(* CoDeSys 2.3.9.28 project: Codesys_Automacao.pro *)
(* Libraries: Standard.lib 27.1.09 11:27:38, Util.lib 27.1.09 11:27:38, IecSfc.lib 24.11.08 08:07:15, SysLibTime.lib 27.1.09 11:27:38, SysTaskInfo.lib 24.11.08 08:07:15, SYSLIBCALLBACK.LIB 27.1.09 11:27:38 *)

(* PLC configuration (modules and I/O channels)
Hexswitch AT %IB0 [HexSwitch] rotary switch 0 = STOP, 1-15 = RUN
IOModules [CPX_MASTER] node 0, in %IB4 out %QB0
  8DI/8DO [CPX-8DI_8DO_Multi_I_O_module_1] node 0, in %IB4 out %QB0 {StringParam = 4,8,1,8,1; ByteParam = 7; ByteParam = 81; ByteParam = 0; ByteParam = 0; ByteParam = 0; ByteParam = 0; ByteParam = 0; IdleStateParam = 0; IdleModeParam = 255; IdleStateParam = 0; IdleModeParam = 255; IdleStateParam = 0; IdleModeParam = 255; IdleStateParam = 0; IdleModeParam = 255}
    AT %IB4 [ByteInput] -
    AT %QB0 [ByteOutput] -
  8DI/8DO [CPX-8DI_8DO_Multi_I_O_module_1] node 1, in %IB8 out %QB4 {StringParam = 4,8,1,8,1; ByteParam = 7; ByteParam = 81; ByteParam = 0; ByteParam = 0; ByteParam = 0; ByteParam = 0; ByteParam = 0; IdleStateParam = 0; IdleModeParam = 255; IdleStateParam = 0; IdleModeParam = 255; IdleStateParam = 0; IdleModeParam = 255; IdleStateParam = 0; IdleModeParam = 255}
    AT %IB8 [ByteInput] -
    AT %QB4 [ByteOutput] -
*)

(* Global variable list: Global_Variables *)
VAR_GLOBAL

	START AT %IX2.0 : BOOL;
	STOP AT %IX2.1 : BOOL;
	B0 AT %IX2.2 : BOOL;

	S1 AT %IX4.4 : BOOL;
	S2 AT %IX4.5 : BOOL;

	S3 AT %IX2.4 : BOOL;
	S4 AT %IX2.5 : BOOL;
	S5 AT %IX2.3 : BOOL;
	S6 AT %IX2.6 : BOOL;
	S7 AT %IX2.7 : BOOL;

	P2_IDA AT %QX2.0 : BOOL;
	P2_VOLTA AT %QX2.1 : BOOL;
	P1 AT %QX2.2 : BOOL;
	P3 AT %QX2.3 : BOOL;



	M1 AT %QX0.0 : BOOL;
	M2 AT %QX0.1 : BOOL;

	LP_1 AT %QX0.2 : BOOL;
	LP_2 AT %QX0.3 : BOOL;
	LP_3 AT %QX0.4 : BOOL;
	AL AT %QX0.5 : BOOL;




	PV_CONT_ENT : INT :=1;
	PV_CONT_SAI : INT :=1;


	M_START : BOOL;
	M_CONT: BOOL;
	M_P1: BOOL;
	M_TEMPERA: BOOL;
	M_2_ENT : BOOL;
	M_2_SAI : BOOL;
	M_ALARME: BOOL;

	MT_1 : BOOL;
	MT_2 : BOOL;
	MT_3 : BOOL;
	MT_4 : BOOL;
	MT_5 : BOOL;

	T_TEMPERA : TON;
	T_ALARME : TON;

    CONT_2_ENT: CTU;
	CONT_2_SAI : CTU;

	BUZZER : APITA_BUZZER;



END_VAR

(* POU PLC_PRG, ST *)
PROGRAM PLC_PRG
VAR

END_VAR
T_TEMPERA(IN:=M_TEMPERA,PT:=T#3S);
T_ALARME(IN:=M_ALARME,PT:=T#5500MS);

CONT_2_ENT(CU:= M_CONT, RESET:= M_2_ENT OR STOP, PV:= PV_CONT_ENT);
CONT_2_SAI(CU:= S7 AND MT_5, RESET:= M_2_SAI OR STOP, PV:= PV_CONT_SAI);

BUZZER(LIGA := AL, DESLIGA := T_ALARME.Q OR START);


IF B0 AND NOT M_START THEN
	PV_CONT_ENT := 1;
	PV_CONT_SAI := 1;
	LP_3 := TRUE;
END_IF

IF NOT B0 AND NOT M_START THEN
	PV_CONT_ENT := 3;
	PV_CONT_SAI := 3;
	LP_3 := FALSE;
END_IF


IF START THEN
	M_START:=TRUE;
	P2_VOLTA:=TRUE;
	LP_1:=TRUE;
END_IF


IF M_START AND S1 THEN
	M1:=TRUE;
	MT_1:=TRUE;
END_IF


IF S2 AND MT_1 THEN
	M_CONT:=TRUE;
	M1:=FALSE;
	MT_1:=FALSE;
ELSE
	M_CONT:= FALSE;
END_IF


IF CONT_2_ENT.Q THEN
	M1:=FALSE;
	P1:=TRUE;
	MT_2:=TRUE;
END_IF


IF S3 AND MT_2 THEN
	P2_IDA:=TRUE;
	P2_VOLTA:=FALSE;
	M_2_ENT:=TRUE;
	MT_2:=FALSE;
	MT_3:=TRUE;
END_IF


IF S4 AND M_2_ENT AND MT_3 THEN
	P2_IDA:=FALSE;
	P2_VOLTA:=TRUE;
	P1:=FALSE;
	MT_3:=FALSE;
	MT_4:=TRUE;
END_IF


IF S5 AND S6 AND MT_4 THEN
	M2:=TRUE;
	M_TEMPERA:=TRUE;
	MT_4:=FALSE;
END_IF


IF T_TEMPERA.Q THEN
	M2:=FALSE;
	P3:=TRUE;
	MT_5:=TRUE;
	LP_2:=TRUE;
END_IF


IF AL THEN
	M_ALARME :=TRUE;
END_IF


IF T_ALARME.Q THEN
	M_ALARME :=FALSE;
END_IF


IF CONT_2_SAI.Q THEN
	AL:=TRUE;
	M_2_ENT:=FALSE;
	M_2_SAI:=TRUE;
	M1:=FALSE;
	M2:=FALSE;

	P1:=FALSE;
	P2_IDA:=FALSE;
	P2_VOLTA:=FALSE;
	P3:=FALSE;

	M_TEMPERA:=FALSE;
	M_START:=FALSE;
	M_CONT:=FALSE;

	MT_1:=FALSE;
	MT_2:=FALSE;
	MT_3:=FALSE;
	MT_4:=FALSE;
	MT_5:=FALSE;

	LP_2:=FALSE;
	LP_1:=FALSE;
ELSE
	M_2_SAI:=FALSE;
END_IF


IF STOP THEN
	M_2_ENT:=FALSE;
	M_2_SAI:=FALSE;
	M_START:=FALSE;
	M1:=FALSE;
	M2:=FALSE;

	P1:=FALSE;
	P2_IDA:=FALSE;
	P2_VOLTA:=TRUE;
	P3:=FALSE;

	M_TEMPERA:=FALSE;
	M_START:=FALSE;
	M_CONT:=FALSE;

	MT_1:=FALSE;
	MT_2:=FALSE;
	MT_3:=FALSE;
	MT_4:=FALSE;
	MT_5:=FALSE;

	LP_2:=FALSE;
	LP_1:=FALSE;
	AL:=FALSE;
END_IF
END_PROGRAM

(* POU APITA_BUZZER, ST *)
FUNCTION_BLOCK APITA_BUZZER
VAR_INPUT
	LIGA : BOOL;
	DESLIGA : BOOL;
END_VAR
VAR_OUTPUT
	SAIDA : BOOL;
END_VAR
VAR
	T1 : TON;
	T2 : TON;
	MEM : BOOL;
END_VAR
T1(IN:=AL, PT:=T#500MS);
T2(IN:= NOT AL, PT:=T#500MS);

IF LIGA AND T1.Q AND MEM THEN
	AL := FALSE;
END_IF


IF NOT LIGA AND T2.Q AND MEM THEN
	AL := TRUE;
END_IF


IF DESLIGA THEN
	MEM := FALSE;
END_IF


IF LIGA THEN
	MEM := TRUE;
END_IF
END_FUNCTION_BLOCK

(* Visualisation screen
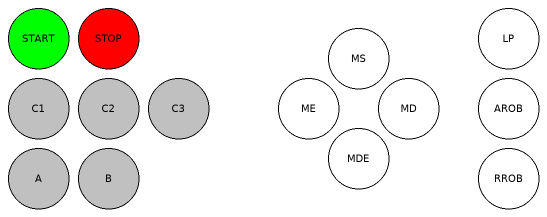
ellipse at (50,120)-(111,181): text "C1"; alarm colour if C1; toggles C1
ellipse at (120,120)-(181,181): text "C2"; alarm colour if C2; toggles C2
ellipse at (190,120)-(251,181): text "C3"; alarm colour if C3; toggles C3
ellipse at (50,50)-(111,111): text "START"; alarm colour if START; taps START
ellipse at (120,50)-(181,111): text "STOP"; alarm colour if STOP; taps STOP
ellipse at (320,120)-(381,181): text "ME"; alarm colour if ME
ellipse at (370,70)-(431,131): text "MS"; alarm colour if MS
ellipse at (370,170)-(431,231): text "MDE"; alarm colour if MDE
ellipse at (420,120)-(481,181): text "MD"; alarm colour if MD
ellipse at (520,50)-(581,111): text "LP"; alarm colour if LP
ellipse at (50,190)-(111,251): text "A"; alarm colour if A; toggles A
ellipse at (120,190)-(181,251): text "B"; alarm colour if B; toggles B
ellipse at (520,120)-(581,181): text "AROB"; alarm colour if AROB
ellipse at (520,190)-(581,251): text "RROB"; alarm colour if RROB
*)

(* Visualisation Simulacao
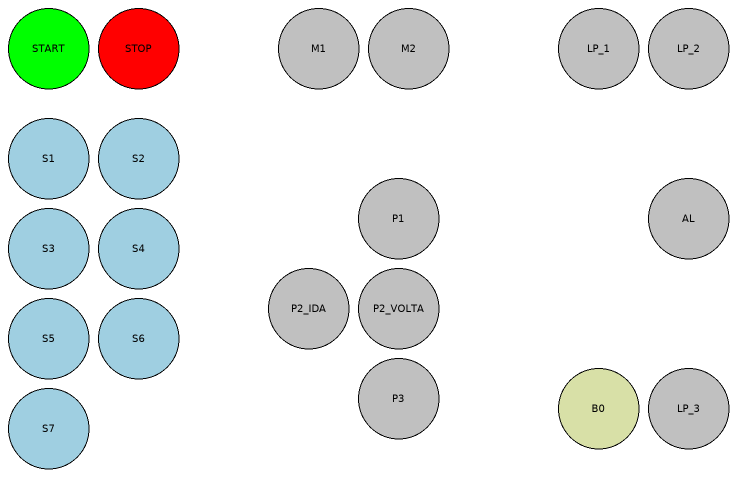
ellipse at (30,30)-(111,111): text "START"; alarm colour if START
ellipse at (120,30)-(201,111): text "STOP"; alarm colour if STOP
ellipse at (30,140)-(111,221): text "S1"; alarm colour if S1
ellipse at (120,140)-(201,221): text "S2"; alarm colour if S2
ellipse at (30,230)-(111,311): text "S3"; alarm colour if S3
ellipse at (120,230)-(201,311): text "S4"; alarm colour if S4
ellipse at (30,320)-(111,401): text "S5"; alarm colour if S5
ellipse at (120,320)-(201,401): text "S6"; alarm colour if S6
ellipse at (300,30)-(381,111): text "M1"; alarm colour if M1
ellipse at (390,30)-(471,111): text "M2"; alarm colour if M2
ellipse at (380,200)-(461,281): text "P1"; alarm colour if P1
ellipse at (380,290)-(461,371): text "P2_VOLTA"; alarm colour if P2_VOLTA
ellipse at (380,380)-(461,461): text "P3"; alarm colour if P3
ellipse at (290,290)-(371,371): text "P2_IDA"; alarm colour if P2_IDA
ellipse at (30,410)-(111,491): text "S7"; alarm colour if S7
ellipse at (670,200)-(751,281): text "AL"; alarm colour if AL
ellipse at (580,30)-(661,111): text "LP_1"; alarm colour if LP_1
ellipse at (670,30)-(751,111): text "LP_2"; alarm colour if LP_2
ellipse at (580,390)-(661,471): text "B0"; alarm colour if B0
ellipse at (670,390)-(751,471): text "LP_3"; alarm colour if LP_3
*)
